FUNCTION MatchesMaterialType : BOOL
VAR_INPUT
	pair : REFERENCE TO PositionMaterials;
	materialPrefix : STRING;
END_VAR
VAR
END_VAR

MatchesMaterialType :=
	FIND(pair.top, materialPrefix) > 0 AND
	FIND(pair.left, materialPrefix) > 0 AND
	FIND(pair.right, materialPrefix) > 0 AND
	FIND(pair.bottom, materialPrefix) > 0 AND
	
	FIND(pair.topLeft, materialPrefix) > 0 AND
	FIND(pair.topRight, materialPrefix) > 0 AND
	FIND(pair.bottomLeft, materialPrefix) > 0 AND
	FIND(pair.bottomRight, materialPrefix) > 0 ;

END_FUNCTION

(* stored: Version 1.1.0.1, ProductVersion 3.1.4024.11
   POU MatchesMaterialType: Id {f5e34751-cdf7-4c56-b6e9-cf2209b10594}, SpecialFunc None *)
